// TwinCAT 3 PLC project FanPlc
// ProgramVersion: 3.1.4024.12
// libraries:
//   Tc2_ModbusRTU, * (Beckhoff Automation GmbH)
//   Tc2_Standard, * (Beckhoff Automation GmbH)
//   Tc2_System, * (Beckhoff Automation GmbH)
//   Tc2_Utilities, * (Beckhoff Automation GmbH)
//   Tc3_Module, * (Beckhoff Automation GmbH)
//   VisuDialogs, * (System)
// project tree:
//   / GlobalTextList.TcGTLO, PlcTask.TcTTO, Visualization Manager.TcVMO (not stored)
//   POUs/ MAIN.TcPOU
//   VISUs/ Visualization.TcVIS
// real-time tasks:
//   TASK PlcTask: cycle T#10ms, priority 20, ADS port 350
// I/O:
//   DEVICE Device 1 (EtherCAT), AmsNetId 5.81.203.152.2.1
//     Term 1 (EK1200) [EK1200-5000 EtherCAT Power supply (2A E-Bus)]
//       Term 2 (EL6021) [EL6021 Interface (RS422/485)]
//       Term 3 (EL9011) [EL9011 End Terminal]
// variable links:
//   FanPlc/FanPlc Instance <-> Device 1 (EtherCAT)/Term 1 (EK1200)/Term 2 (EL6021)
//     PlcTask Inputs/MAIN.mbMaster.InData @bit {16..184 step 8} <-> COM TxPDO-Map Inputs/Data In {0..21}  (22 links)
//     PlcTask Inputs/MAIN.mbMaster.InData <-> COM TxPDO-Map Inputs/Status
//     PlcTask Outputs/MAIN.mbMaster.OutData <-> COM RxPDO-Map Outputs/Ctrl
//     PlcTask Outputs/MAIN.mbMaster.OutData @bit {16..184 step 8} <-> COM RxPDO-Map Outputs/Data Out {0..21}  (22 links)

CONFIGURATION FanPlc
    RESOURCE PLC ON TwinCAT3
        TASK PlcTask(INTERVAL := T#10ms, PRIORITY := 20);
        PROGRAM MAIN WITH PlcTask : MAIN;
    END_RESOURCE
END_CONFIGURATION

// ---- POUs/MAIN.TcPOU
PROGRAM MAIN
VAR
	state		: UINT := 0;
	
	mbMaster	: ModbusRtuMaster_KL6x22B;
	mbUnit		: BYTE := 1;
	mbQuantity	: UINT := 1;
	mbErrorFlag	: BOOL;
	mbErrorId	: MODBUS_ERRORS;
	mbExecute	: BOOL;
	mbBusy		: BOOL;
	mbBytesRec	: UINT;
	
	mbReadAddr	: UINT;
	mbWriteAddr : WORD;
	mbReadData	: WORD;
	mbWriteData : WORD;
	
END_VAR


CASE state OF
0: // init
	mbExecute := TRUE;
1: // read input register
	mbMaster.ReadInputRegs(
		UnitID:= mbUnit, 
		Quantity:= mbQuantity, 
		MBAddr:= mbReadAddr, 
		cbLength:= SIZEOF(mbReadData), 
		pMemoryAddr:= ADR(mbReadData), 
		Execute:= mbExecute, 
		Timeout:= T#1S, 
		BUSY=> mbBusy, 
		Error=> mbErrorFlag, 
		ErrorId=> mbErrorId, 
		cbRead=> mbBytesRec);
	// if busy, turn off exec; if not busy, flip exec
	IF mbBusy = TRUE THEN
		mbExecute := FALSE;
	//ELSE
	//	mbExecute := mbExecute XOR TRUE;
	END_IF
	
2: // read register
	mbMaster.ReadRegs(
		UnitID:= mbUnit, 
		Quantity:= mbQuantity, 
		MBAddr:= mbReadAddr, 
		cbLength:= SIZEOF(mbReadData), 
		pMemoryAddr:= ADR(mbReadData), 
		Execute:= mbExecute, 
		Timeout:= T#1S, 
		BUSY=> mbBusy, 
		Error=> mbErrorFlag, 
		ErrorId=> mbErrorId, 
		cbRead=> mbBytesRec);
	// if busy, turn off exec; if not busy, flip exec
	IF mbBusy = TRUE THEN
		mbExecute := FALSE;
	//ELSE
	//	mbExecute := mbExecute XOR TRUE;
	END_IF
	
3: // write register
	mbMaster.WriteSingleRegister(
		UnitID:= mbUnit, 
		Quantity:= mbQuantity, 
		MBAddr:= mbReadAddr, 
		cbLength:= SIZEOF(mbWriteData), 
		pMemoryAddr:= ADR(mbWriteData), 
		Execute:= mbExecute, 
		Timeout:= T#1S, 
		BUSY=> mbBusy, 
		Error=> mbErrorFlag, 
		ErrorId=> mbErrorId, 
		cbRead=> mbBytesRec);
		
	// if busy, turn off exec; if not busy, flip exec
	IF mbBusy = TRUE THEN
		mbExecute := FALSE;
	//ELSE
	//	mbExecute := mbExecute XOR TRUE;
	END_IF
	
END_CASE

END_PROGRAM

// ---- GlobalTextList.TcGTLO
TEXTLIST GlobalTextList
  486 = '%h'
  833 = '%s'
  795 = '%X'
  129 = 'Address'
  223 = 'Data'
  285 = 'Init'
  572 = 'Read'
  102 = 'Read Reg'
  82 = 'ReadInputReg'
  783 = 'ReadReg'
  86 = 'Test %d'
  70 = 'Test %X'
  15 = 'Write'
  220 = 'Write\t'
  8 = 'WriteReg'
END_TEXTLIST

// ---- VISUs/Visualization.TcVIS
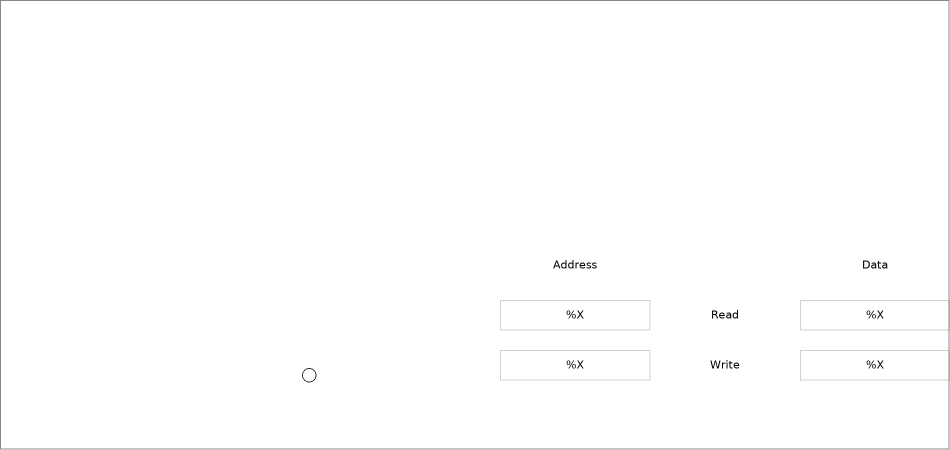
VISUALIZATION Visualization  // 950x450
    RadioButton (300,300 150x150), variable: MAIN.state
        Areas[0]: Text=Init
        Areas[1]: Text=ReadInputReg
        Areas[2]: Text=ReadReg
        Areas[3]: Text=WriteReg
    Textfield (500,300 150x30), "%X", text variable: MAIN.mbReadAddr
        OnMouseClick: write the text variable via Default, format %X
    Label (650,300 150x30), "Read"
    Label (500,250 150x30), "Address"
    Label (800,250 150x30), "Data"
    Textfield (800,300 150x30), "%X", text variable: MAIN.mbReadData
    Textfield (800,350 150x30), "%X", text variable: MAIN.mbWriteData
        OnMouseClick: write the text variable via Default
    Textfield (500,350 150x30), "%X", text variable: MAIN.mbWriteAddr
        OnMouseClick: write the text variable via Default, format %X
    Label (650,350 150x30), "Write"
END_VISUALIZATION
